(* Logix 5000 project; controller Lab7_1 5069-L306ERM rev 35.16; software revision 35.00 *)

TASK MainTask (continuous, watchdog 500 ms) : MainProgram

MODULES
   Local : 5069-L306ERM (5069 0, rev 35.16)
      IOHub : vendor 1 type 7 code 358 (Ethernet 192.168.110.5, rev 1.1, Output RPI 20 ms)
END_MODULES

PROGRAM MainProgram   (* main routine MainRoutine *)
VAR
   countDown2 : COUNTER := (PRE := 2);
   countDown3 : COUNTER := (PRE := 3);
   counter_0 : COUNTER;
   counter_2 : COUNTER;
   displayTimer : TIMER := (PRE := 5000);
   Dummy : BOOL;
   enable_1_sec : BOOL;
   enable_3_sec : BOOL;
   flash1 : BOOL;
   flash1TOF : TIMER := (PRE := 1000);
   flash2 : BOOL;
   flash2TOF : TIMER := (PRE := 1000);
   flash2TON : TIMER := (PRE := 2000);
   flash3 : BOOL;
   flash3TOF : TIMER := (PRE := 1000);
   flash3TON : TIMER := (PRE := 2000);
   flash_1 : BOOL;
   flash_1TOF : TIMER := (PRE := 1000);
   HOLD : BOOL;
   HOLD2 : BOOL;
   timer : TIMER := (PRE := 1000);
   timer_1_sec : TIMER := (PRE := 1000);
   timer_3_sec : TIMER := (PRE := 3000);
END_VAR

ROUTINE MainRoutine   (* ladder *)
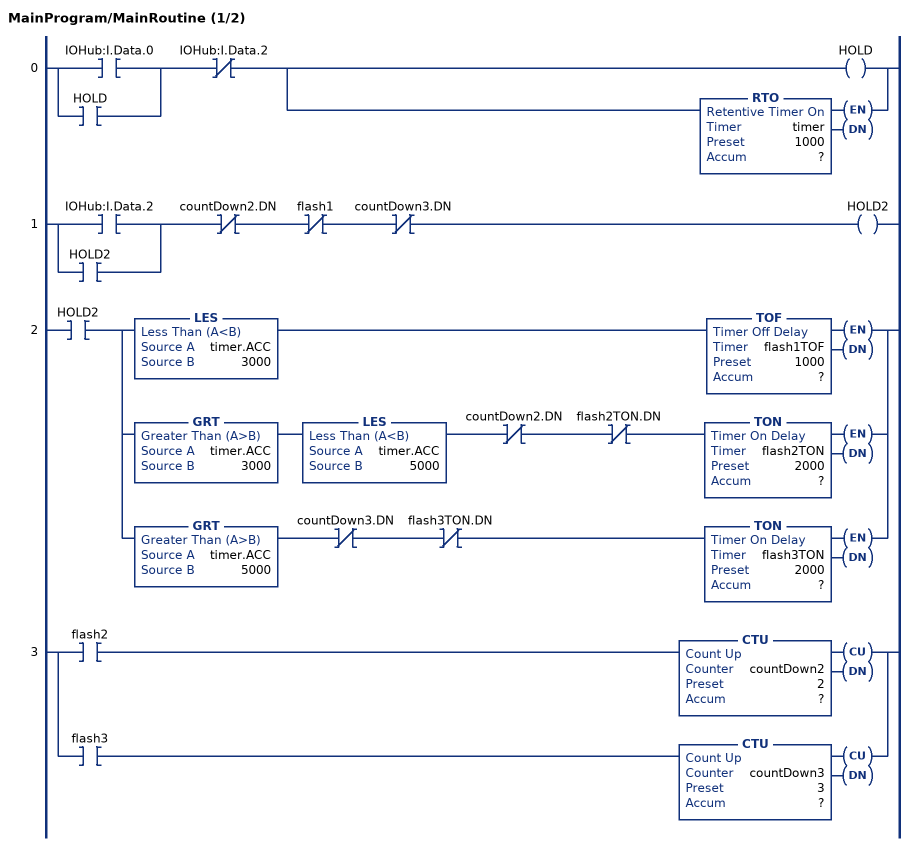
   0: [XIC(IOHub:I.Data.0) ,XIC(HOLD) ]XIO(IOHub:I.Data.2)[OTE(HOLD) ,RTO(timer,?,?) ];
   1: [XIC(IOHub:I.Data.2) ,XIC(HOLD2) ]XIO(countDown2.DN)XIO(flash1)XIO(countDown3.DN)OTE(HOLD2);
   2: XIC(HOLD2)[LES(timer.ACC,3000) TOF(flash1TOF,?,?) ,[GRT(timer.ACC,3000) LES(timer.ACC,5000) XIO(countDown2.DN) XIO(flash2TON.DN) TON(flash2TON,?,?) ,GRT(timer.ACC,5000) XIO(countDown3.DN) XIO(flash3TON.DN) TON(flash3TON,?,?) ] ];
   3: [XIC(flash2) CTU(countDown2,?,?) ,XIC(flash3) CTU(countDown3,?,?) ];
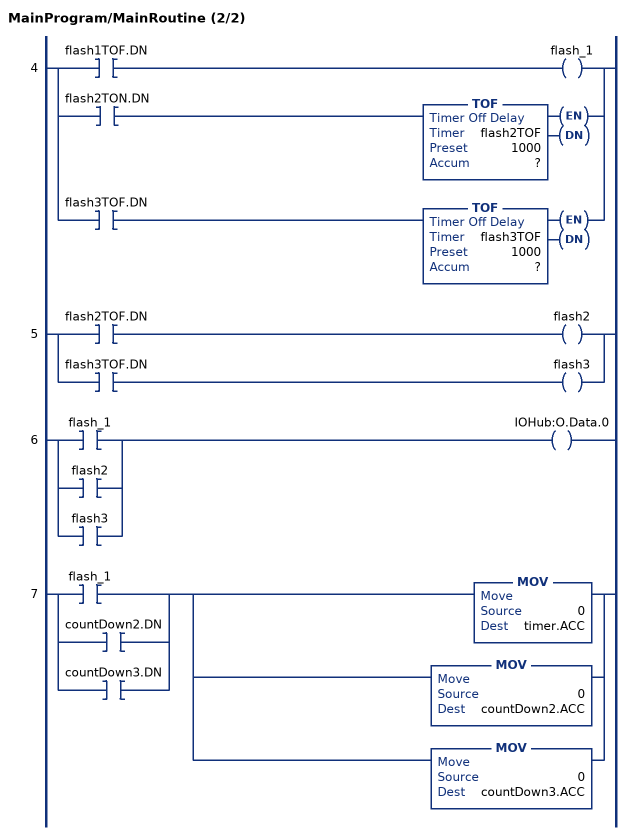
   4: [XIC(flash1TOF.DN) OTE(flash_1) ,[XIC(flash2TON.DN) TOF(flash2TOF,?,?) ,XIC(flash3TOF.DN) TOF(flash3TOF,?,?) ] ];
   5: [XIC(flash2TOF.DN) OTE(flash2) ,XIC(flash3TOF.DN) OTE(flash3) ];
   6: [XIC(flash_1) ,[XIC(flash2) ,XIC(flash3) ] ]OTE(IOHub:O.Data.0);
   7: [XIC(flash_1) ,[XIC(countDown2.DN) ,XIC(countDown3.DN) ] ][MOV(0,timer.ACC) ,[MOV(0,countDown2.ACC) ,MOV(0,countDown3.ACC) ] ];
END_ROUTINE
END_PROGRAM
